FUNCTION_BLOCK FB_LD_PressDemoAuto EXTENDS FB_SequenceBase
VAR
    _partReady, _airReady, _startReady, _stop, _doStep, _processed, _endCycle, _dummy : BOOL;
    _dwellTwoHandHeld : BOOL;          // N220 named wait: two-hand held through the dwell
    _decisionRequest : ST_DecisionRequest;   // §6.11 not-reached confirmation
    _answer : INT;
    _ramReached, _failureConfirmed : BOOL;   // N200/N210 named waits
    _twoHandHeldDuringClose : BOOL;          // N180 named wait
    _closeAbortWarned : BOOL;                // N180 §6.9(e) message result
    _ramFailureReported : BOOL;              // N200 §6.9(e) message result
    _partInMachine : BOOL;                   // §3.16.3 the part is already received
    _partDispositioned : BOOL;               // N260 already set the verdict
    _traceAccepted, _recordAccepted, _partProcessed : BOOL;
    {attribute 'OPC.UA.DA' := '0'}
    _pressRam : REFERENCE TO FB_CylinderCM;
    {attribute 'OPC.UA.DA' := '0'}
    _door : REFERENCE TO FB_CylinderCM;
    {attribute 'OPC.UA.DA' := '0'}
    _partSlide : REFERENCE TO FB_CylinderCM;
    {attribute 'OPC.UA.DA' := '0'}
    _twoHand : REFERENCE TO FB_TwoHandStartCM;
    {attribute 'OPC.UA.DA' := '0'}
    _partPresentSensor : REFERENCE TO FB_DigitalInputCM;
    {attribute 'OPC.UA.DA' := '0'}
    _airPressureMonitor : REFERENCE TO FB_AirPressureMonitorCM;
    {attribute 'OPC.UA.DA' := '0'}
    _parCfg : REFERENCE TO ST_PneumaticPressParCfg;
    // §3.8a - the cell's own policy, referenced like _parCfg.
    {attribute 'OPC.UA.DA' := '0'}
    _stationCfg : REFERENCE TO ST_PneumaticPressStationCfg;
    {attribute 'OPC.UA.DA' := '0'}
    _outCmd : REFERENCE TO ST_PneumaticPressOutCmd;
    {attribute 'OPC.UA.DA' := '0'}
    _startLatched : REFERENCE TO BOOL;
    {attribute 'OPC.UA.DA' := '0'}
    _loadPosition : FB_PressDemoLoadPosition;
END_VAR
VAR // added by the converter: edge detectors and wires of the graphical bodies
    _w1, _w2, _w3, _w4, _w5, _w6, _w7, _w8, _w9, _w10, _w11, _w12, _w13, _w14, _w15, _w16, _w17, _w18, _w19, _w20, _w21, _w22, _w23, _w24, _w25, _w26, _w27, _w28, _w29, _w30 : BOOL;
END_VAR

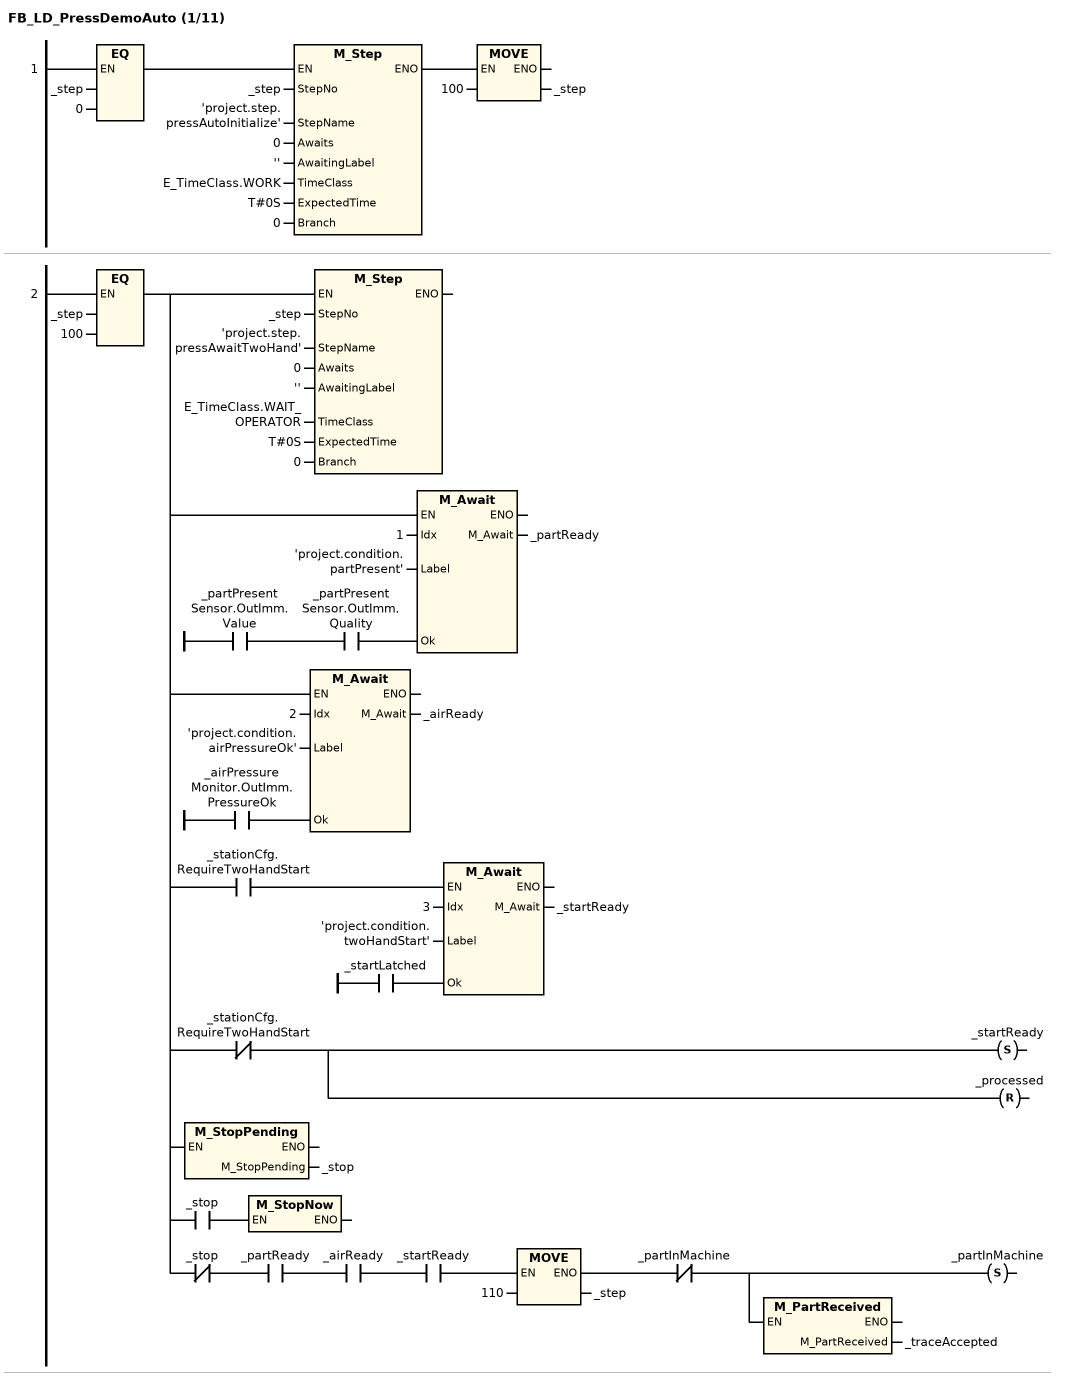
// NETWORK 1
_w1 := _step = 0;
IF _w1 THEN
    M_Step(StepNo := _step, StepName := 'project.step.pressAutoInitialize', Awaits := 0, AwaitingLabel := '', TimeClass := E_TimeClass.WORK, ExpectedTime := T#0S, Branch := 0);
END_IF
IF _w1 THEN _step := 100; END_IF

// NETWORK 2
_w2 := _step = 100;
IF _w2 THEN
    M_Step(StepNo := _step, StepName := 'project.step.pressAwaitTwoHand', Awaits := 0, AwaitingLabel := '', TimeClass := E_TimeClass.WAIT_OPERATOR, ExpectedTime := T#0S, Branch := 0);
END_IF
IF _w2 THEN
    _partReady := M_Await(Idx := 1, Label := 'project.condition.partPresent', Ok := _partPresentSensor.OutImm.Value AND _partPresentSensor.OutImm.Quality);
END_IF
IF _w2 THEN
    _airReady := M_Await(Idx := 2, Label := 'project.condition.airPressureOk', Ok := _airPressureMonitor.OutImm.PressureOk);
END_IF
IF _w2 AND _stationCfg.RequireTwoHandStart THEN
    _startReady := M_Await(Idx := 3, Label := 'project.condition.twoHandStart', Ok := _startLatched);
END_IF
_w3 := _w2 AND NOT _stationCfg.RequireTwoHandStart;
_startReady S= _w3;
_processed R= _w3;
IF _w2 THEN _stop := M_StopPending(); END_IF
IF _w2 AND _stop THEN M_StopNow(); END_IF
IF _w2 AND NOT _stop AND _partReady AND _airReady AND _startReady THEN _step := 110; END_IF
_w4 := (_w2 AND NOT _stop AND _partReady AND _airReady AND _startReady) AND NOT _partInMachine;
_partInMachine S= _w4;
IF _w4 THEN _traceAccepted := M_PartReceived(); END_IF

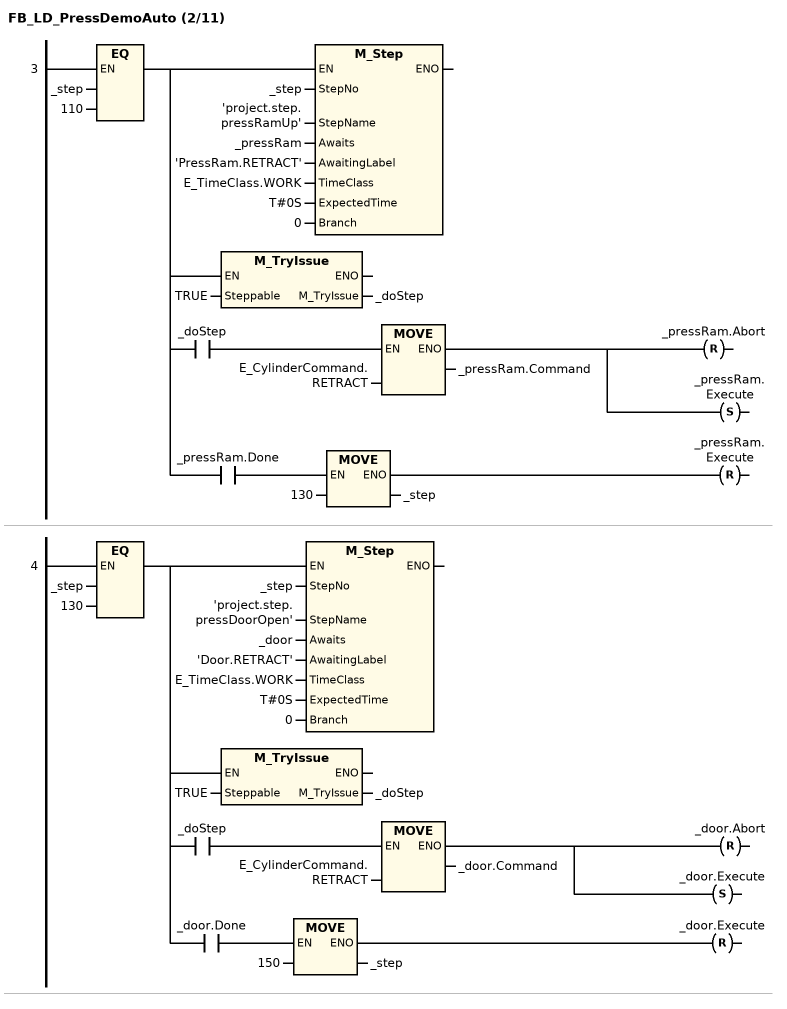
// NETWORK 3
_w5 := _step = 110;
IF _w5 THEN
    M_Step(StepNo := _step, StepName := 'project.step.pressRamUp', Awaits := _pressRam, AwaitingLabel := 'PressRam.RETRACT', TimeClass := E_TimeClass.WORK, ExpectedTime := T#0S, Branch := 0);
END_IF
IF _w5 THEN _doStep := M_TryIssue(Steppable := TRUE); END_IF
IF _w5 AND _doStep THEN _pressRam.Command := E_CylinderCommand.RETRACT; END_IF
_w6 := _w5 AND _doStep;
_pressRam.Abort R= _w6;
_pressRam.Execute S= _w6;
IF _w5 AND _pressRam.Done THEN _step := 130; END_IF
_pressRam.Execute R= _w5 AND _pressRam.Done;

// NETWORK 4
_w7 := _step = 130;
IF _w7 THEN
    M_Step(StepNo := _step, StepName := 'project.step.pressDoorOpen', Awaits := _door, AwaitingLabel := 'Door.RETRACT', TimeClass := E_TimeClass.WORK, ExpectedTime := T#0S, Branch := 0);
END_IF
IF _w7 THEN _doStep := M_TryIssue(Steppable := TRUE); END_IF
IF _w7 AND _doStep THEN _door.Command := E_CylinderCommand.RETRACT; END_IF
_w8 := _w7 AND _doStep;
_door.Abort R= _w8;
_door.Execute S= _w8;
IF _w7 AND _door.Done THEN _step := 150; END_IF
_door.Execute R= _w7 AND _door.Done;

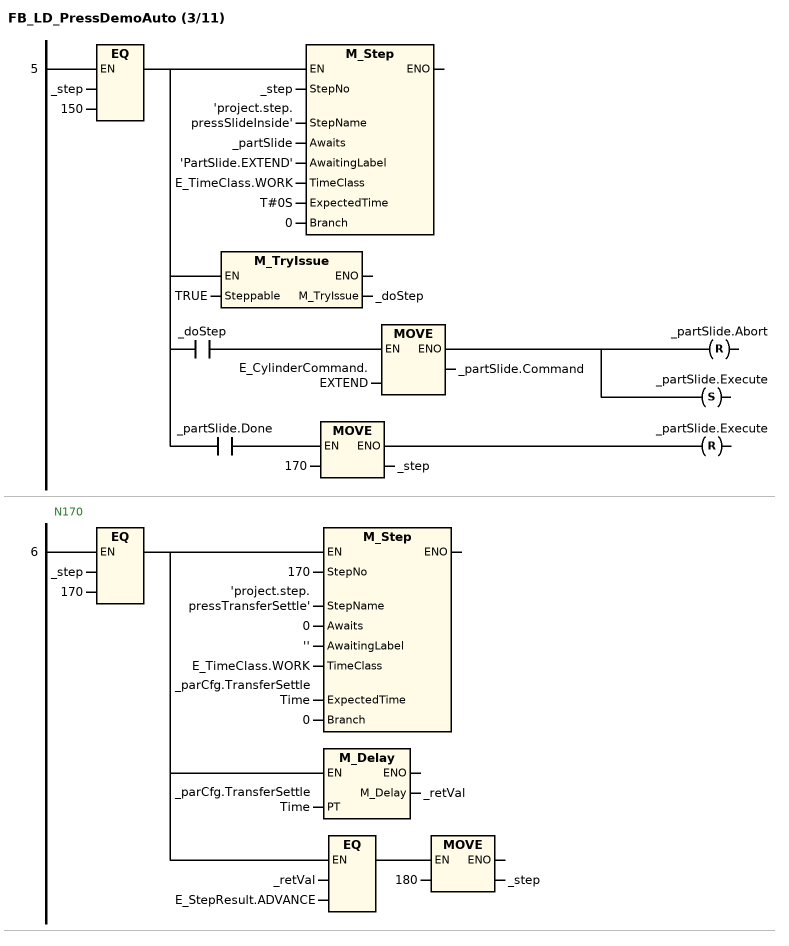
// NETWORK 5
_w9 := _step = 150;
IF _w9 THEN
    M_Step(StepNo := _step, StepName := 'project.step.pressSlideInside', Awaits := _partSlide, AwaitingLabel := 'PartSlide.EXTEND', TimeClass := E_TimeClass.WORK, ExpectedTime := T#0S, Branch := 0);
END_IF
IF _w9 THEN _doStep := M_TryIssue(Steppable := TRUE); END_IF
IF _w9 AND _doStep THEN _partSlide.Command := E_CylinderCommand.EXTEND; END_IF
_w10 := _w9 AND _doStep;
_partSlide.Abort R= _w10;
_partSlide.Execute S= _w10;
IF _w9 AND _partSlide.Done THEN _step := 170; END_IF
_partSlide.Execute R= _w9 AND _partSlide.Done;

// NETWORK 6
// N170
_w11 := _step = 170;
IF _w11 THEN
    M_Step(StepNo := 170, StepName := 'project.step.pressTransferSettle', Awaits := 0, AwaitingLabel := '', TimeClass := E_TimeClass.WORK, ExpectedTime := _parCfg.TransferSettleTime, Branch := 0);
END_IF
IF _w11 THEN _retVal := M_Delay(PT := _parCfg.TransferSettleTime); END_IF
IF _w11 AND _retVal = E_StepResult.ADVANCE THEN _step := 180; END_IF

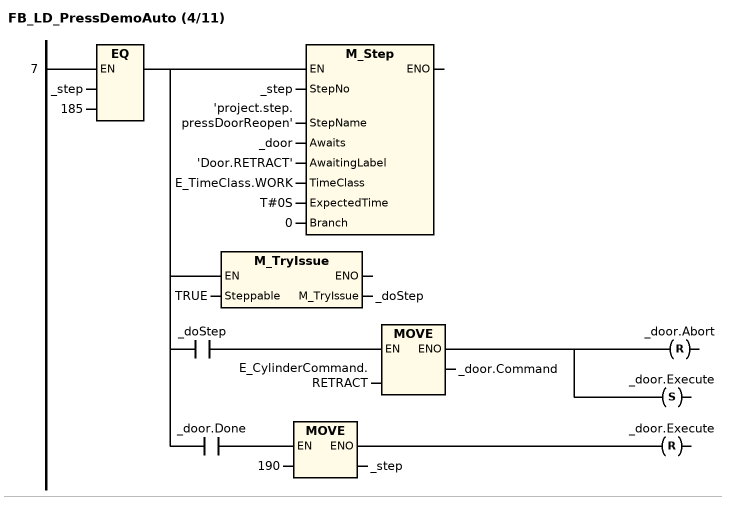
// NETWORK 7
_w12 := _step = 185;
IF _w12 THEN
    M_Step(StepNo := _step, StepName := 'project.step.pressDoorReopen', Awaits := _door, AwaitingLabel := 'Door.RETRACT', TimeClass := E_TimeClass.WORK, ExpectedTime := T#0S, Branch := 0);
END_IF
IF _w12 THEN _doStep := M_TryIssue(Steppable := TRUE); END_IF
IF _w12 AND _doStep THEN _door.Command := E_CylinderCommand.RETRACT; END_IF
_w13 := _w12 AND _doStep;
_door.Abort R= _w13;
_door.Execute S= _w13;
IF _w12 AND _door.Done THEN _step := 190; END_IF
_door.Execute R= _w12 AND _door.Done;

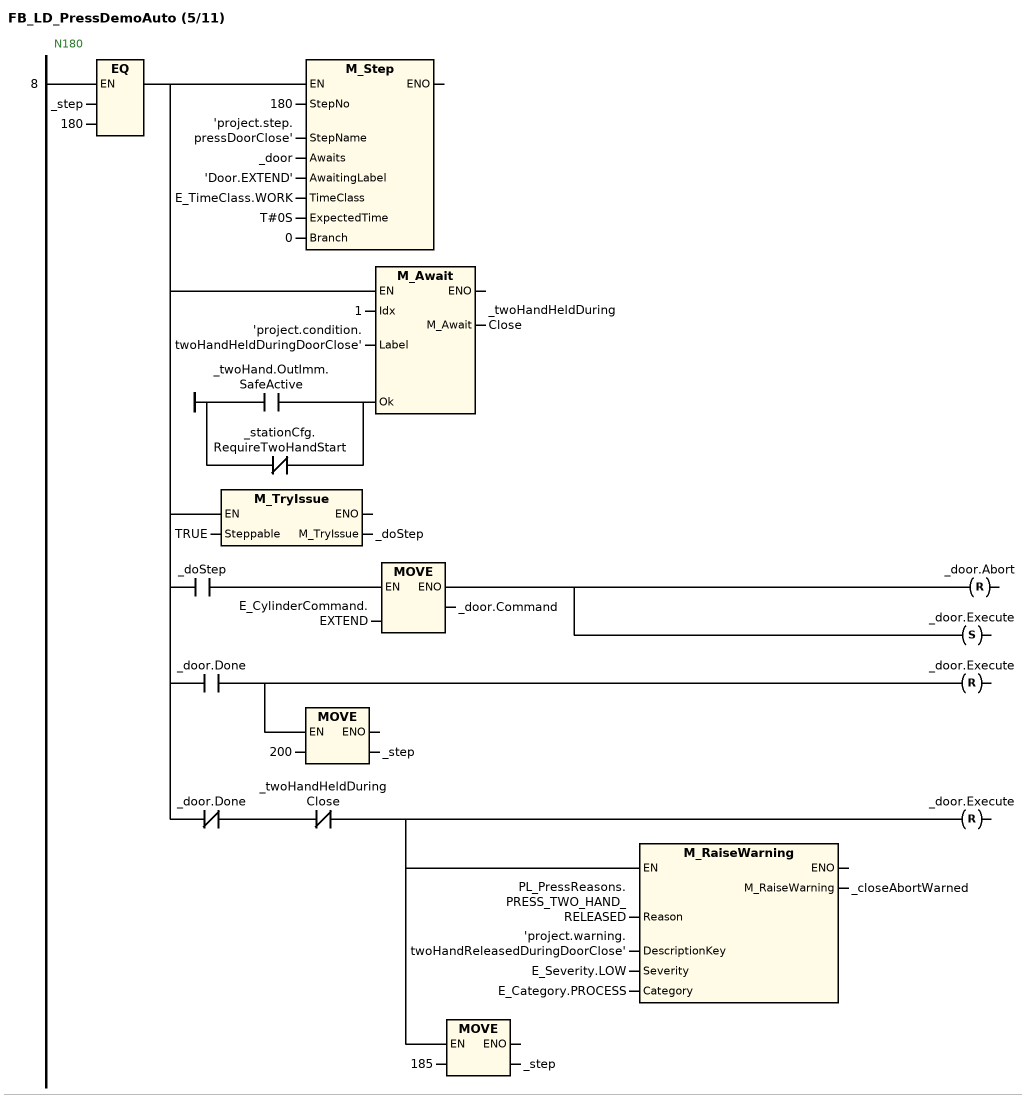
// NETWORK 8
// N180
_w14 := _step = 180;
IF _w14 THEN
    M_Step(StepNo := 180, StepName := 'project.step.pressDoorClose', Awaits := _door, AwaitingLabel := 'Door.EXTEND', TimeClass := E_TimeClass.WORK, ExpectedTime := T#0S, Branch := 0);
END_IF
IF _w14 THEN
    _twoHandHeldDuringClose := M_Await(Idx := 1, Label := 'project.condition.twoHandHeldDuringDoorClose', Ok := _twoHand.OutImm.SafeActive OR NOT _stationCfg.RequireTwoHandStart);
END_IF
IF _w14 THEN _doStep := M_TryIssue(Steppable := TRUE); END_IF
IF _w14 AND _doStep THEN _door.Command := E_CylinderCommand.EXTEND; END_IF
_w15 := _w14 AND _doStep;
_door.Abort R= _w15;
_door.Execute S= _w15;
_w16 := _w14 AND _door.Done;
_door.Execute R= _w16;
IF _w16 THEN _step := 200; END_IF
_w17 := _w14 AND NOT _door.Done AND NOT _twoHandHeldDuringClose;
_door.Execute R= _w17;
IF _w17 THEN
    _closeAbortWarned := M_RaiseWarning(Reason := PL_PressReasons.PRESS_TWO_HAND_RELEASED, DescriptionKey := 'project.warning.twoHandReleasedDuringDoorClose', Severity := E_Severity.LOW, Category := E_Category.PROCESS);
END_IF
IF _w17 THEN _step := 185; END_IF

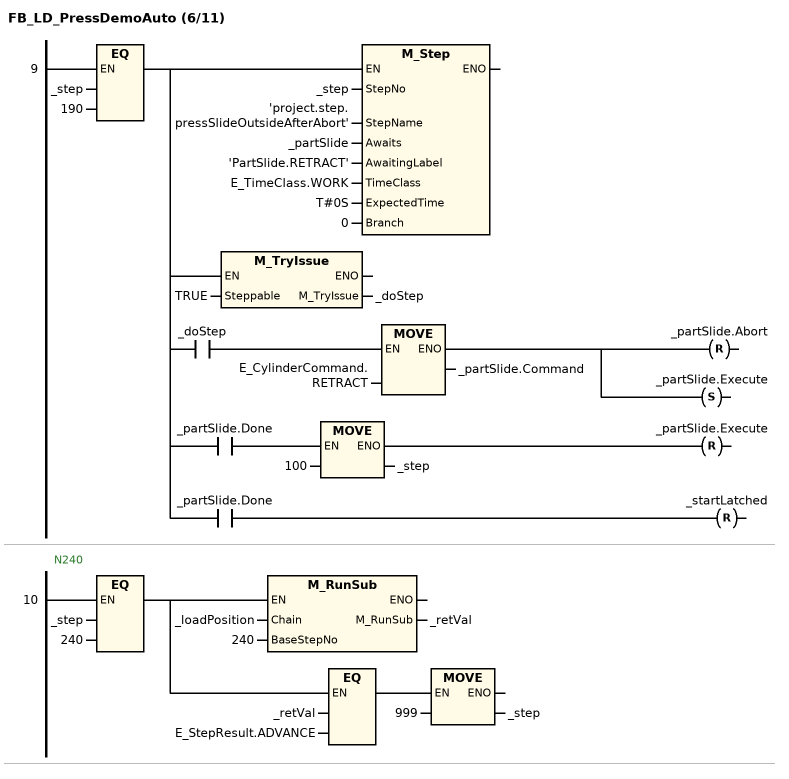
// NETWORK 9
_w18 := _step = 190;
IF _w18 THEN
    M_Step(StepNo := _step, StepName := 'project.step.pressSlideOutsideAfterAbort', Awaits := _partSlide, AwaitingLabel := 'PartSlide.RETRACT', TimeClass := E_TimeClass.WORK, ExpectedTime := T#0S, Branch := 0);
END_IF
IF _w18 THEN _doStep := M_TryIssue(Steppable := TRUE); END_IF
IF _w18 AND _doStep THEN _partSlide.Command := E_CylinderCommand.RETRACT; END_IF
_w19 := _w18 AND _doStep;
_partSlide.Abort R= _w19;
_partSlide.Execute S= _w19;
IF _w18 AND _partSlide.Done THEN _step := 100; END_IF
_partSlide.Execute R= _w18 AND _partSlide.Done;
_startLatched R= _w18 AND _partSlide.Done;

// NETWORK 10
// N240
_w20 := _step = 240;
IF _w20 THEN _retVal := M_RunSub(Chain := _loadPosition, BaseStepNo := 240); END_IF
IF _w20 AND _retVal = E_StepResult.ADVANCE THEN _step := 999; END_IF

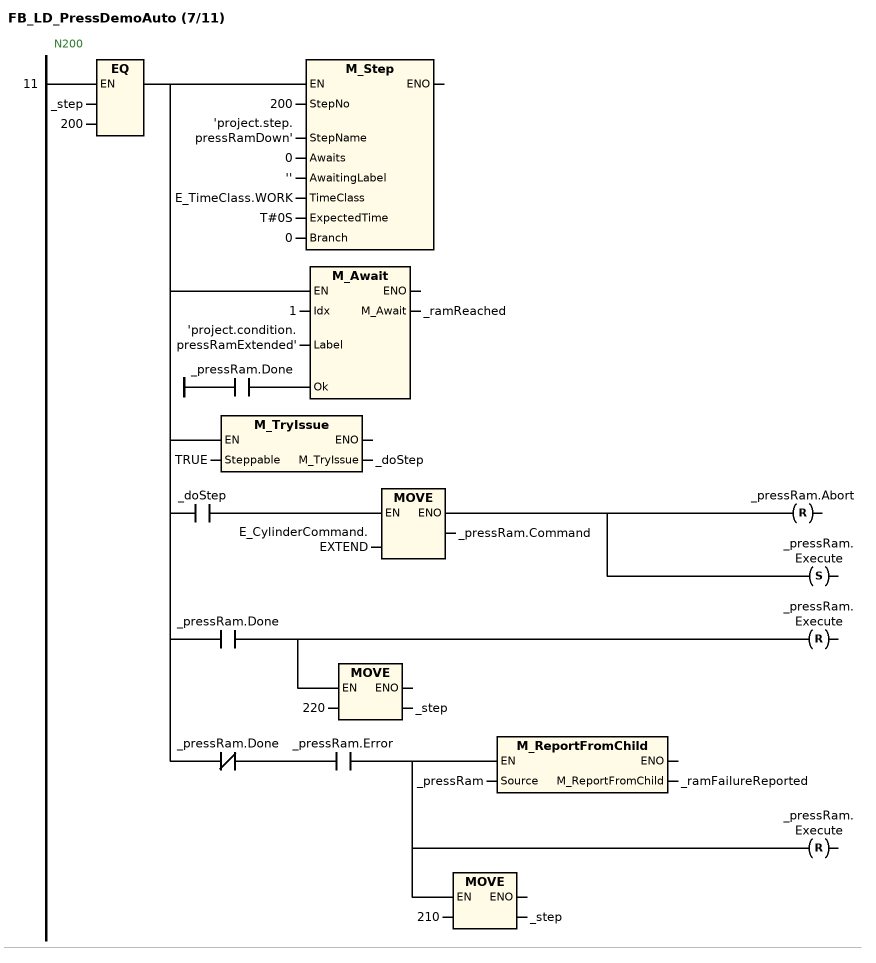
// NETWORK 11
// N200
_w21 := _step = 200;
IF _w21 THEN
    M_Step(StepNo := 200, StepName := 'project.step.pressRamDown', Awaits := 0, AwaitingLabel := '', TimeClass := E_TimeClass.WORK, ExpectedTime := T#0S, Branch := 0);
END_IF
IF _w21 THEN
    _ramReached := M_Await(Idx := 1, Label := 'project.condition.pressRamExtended', Ok := _pressRam.Done);
END_IF
IF _w21 THEN _doStep := M_TryIssue(Steppable := TRUE); END_IF
IF _w21 AND _doStep THEN _pressRam.Command := E_CylinderCommand.EXTEND; END_IF
_w22 := _w21 AND _doStep;
_pressRam.Abort R= _w22;
_pressRam.Execute S= _w22;
_w23 := _w21 AND _pressRam.Done;
_pressRam.Execute R= _w23;
IF _w23 THEN _step := 220; END_IF
_w24 := _w21 AND NOT _pressRam.Done AND _pressRam.Error;
IF _w24 THEN _ramFailureReported := M_ReportFromChild(Source := _pressRam); END_IF
_pressRam.Execute R= _w24;
IF _w24 THEN _step := 210; END_IF

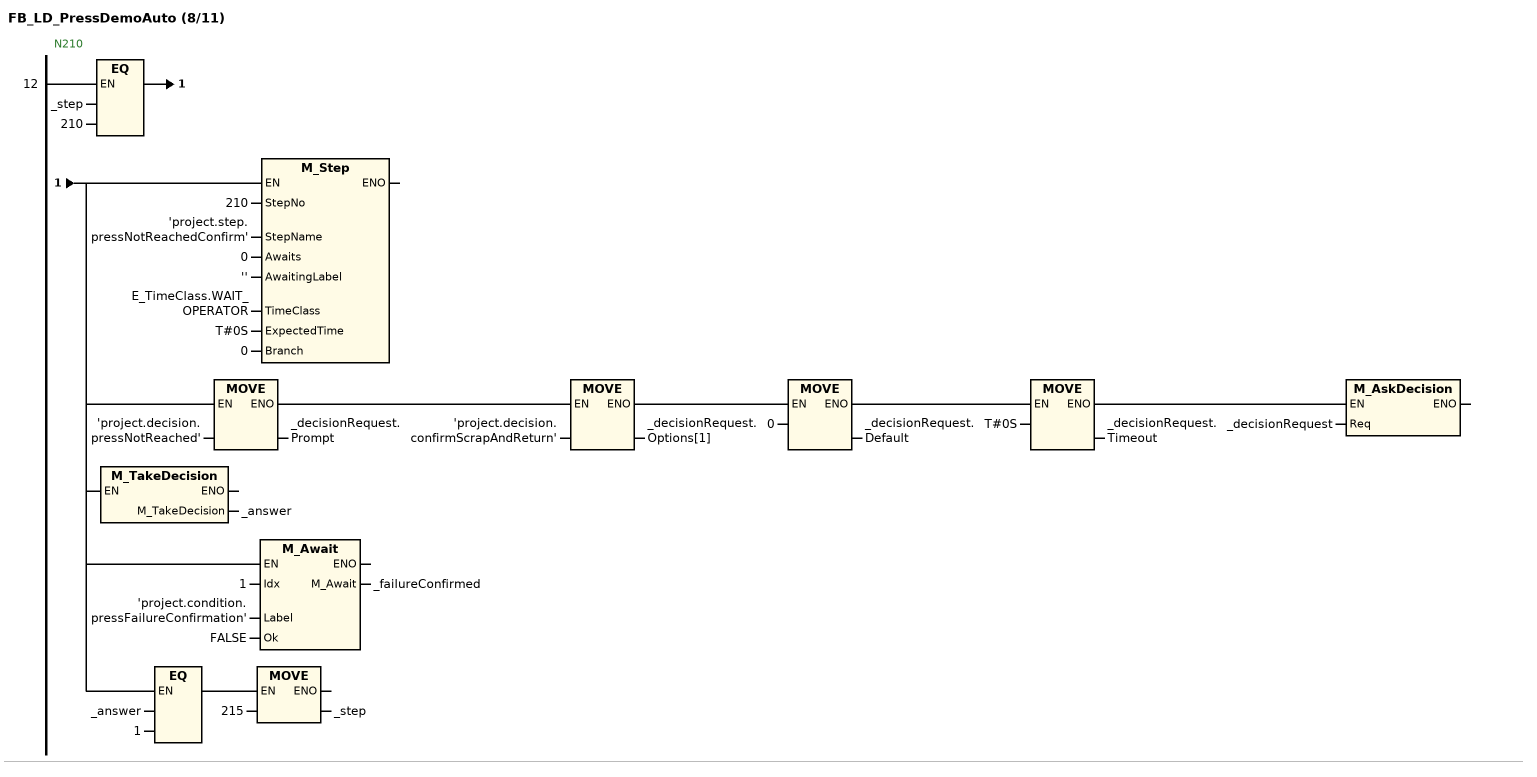
// NETWORK 12
// N210
_w25 := _step = 210;
IF _w25 THEN
    M_Step(StepNo := 210, StepName := 'project.step.pressNotReachedConfirm', Awaits := 0, AwaitingLabel := '', TimeClass := E_TimeClass.WAIT_OPERATOR, ExpectedTime := T#0S, Branch := 0);
END_IF
IF _w25 THEN _decisionRequest.Prompt := 'project.decision.pressNotReached'; END_IF
IF _w25 THEN _decisionRequest.Options[1] := 'project.decision.confirmScrapAndReturn'; END_IF
IF _w25 THEN _decisionRequest.Default := 0; END_IF
IF _w25 THEN _decisionRequest.Timeout := T#0S; END_IF
IF _w25 THEN M_AskDecision(Req := _decisionRequest); END_IF
IF _w25 THEN _answer := M_TakeDecision(); END_IF
IF _w25 THEN
    _failureConfirmed := M_Await(Idx := 1, Label := 'project.condition.pressFailureConfirmation', Ok := FALSE);
END_IF
IF _w25 AND _answer = 1 THEN _step := 215; END_IF

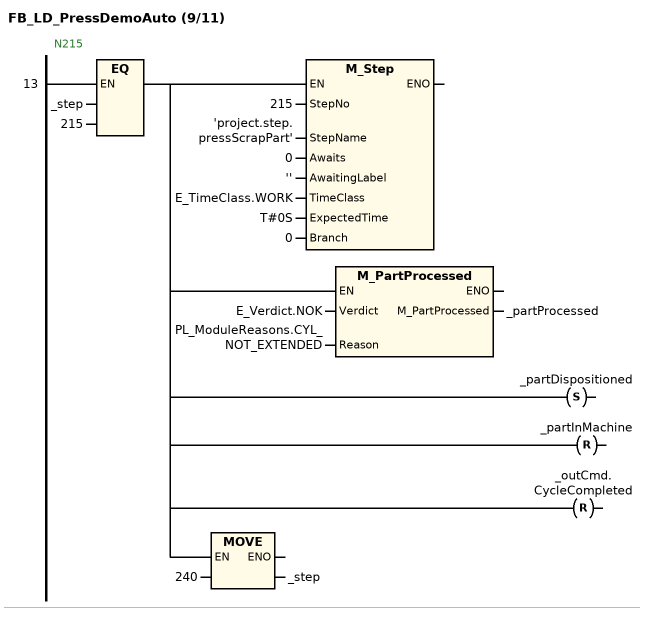
// NETWORK 13
// N215
_w26 := _step = 215;
IF _w26 THEN
    M_Step(StepNo := 215, StepName := 'project.step.pressScrapPart', Awaits := 0, AwaitingLabel := '', TimeClass := E_TimeClass.WORK, ExpectedTime := T#0S, Branch := 0);
END_IF
IF _w26 THEN
    _partProcessed := M_PartProcessed(Verdict := E_Verdict.NOK, Reason := PL_ModuleReasons.CYL_NOT_EXTENDED);
END_IF
_partDispositioned S= _w26;
_partInMachine R= _w26;
_outCmd.CycleCompleted R= _w26;
IF _w26 THEN _step := 240; END_IF

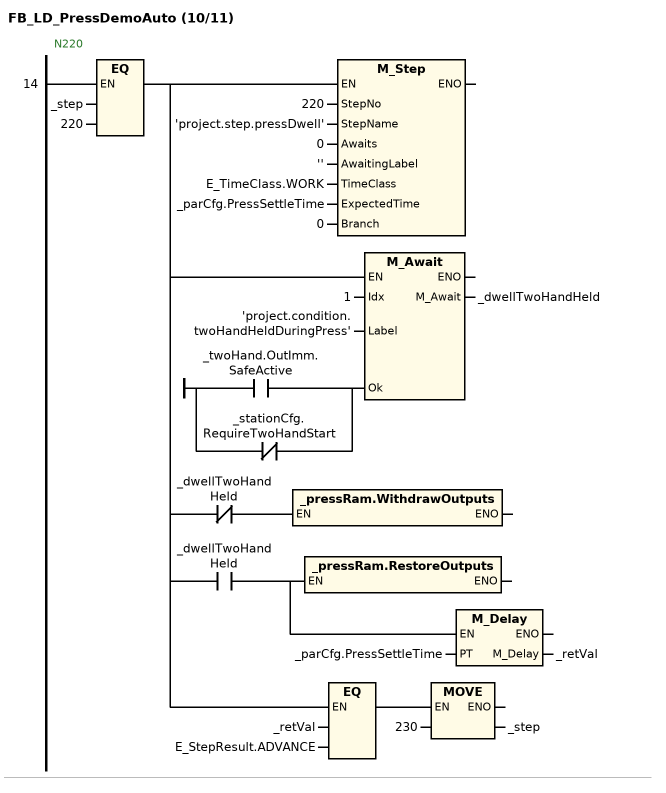
// NETWORK 14
// N220
_w27 := _step = 220;
IF _w27 THEN
    M_Step(StepNo := 220, StepName := 'project.step.pressDwell', Awaits := 0, AwaitingLabel := '', TimeClass := E_TimeClass.WORK, ExpectedTime := _parCfg.PressSettleTime, Branch := 0);
END_IF
IF _w27 THEN
    _dwellTwoHandHeld := M_Await(Idx := 1, Label := 'project.condition.twoHandHeldDuringPress', Ok := _twoHand.OutImm.SafeActive OR NOT _stationCfg.RequireTwoHandStart);
END_IF
IF _w27 AND NOT _dwellTwoHandHeld THEN _pressRam.WithdrawOutputs(); END_IF
_w28 := _w27 AND _dwellTwoHandHeld;
IF _w28 THEN _pressRam.RestoreOutputs(); END_IF
IF _w28 THEN _retVal := M_Delay(PT := _parCfg.PressSettleTime); END_IF
IF _w27 AND _retVal = E_StepResult.ADVANCE THEN _step := 230; END_IF

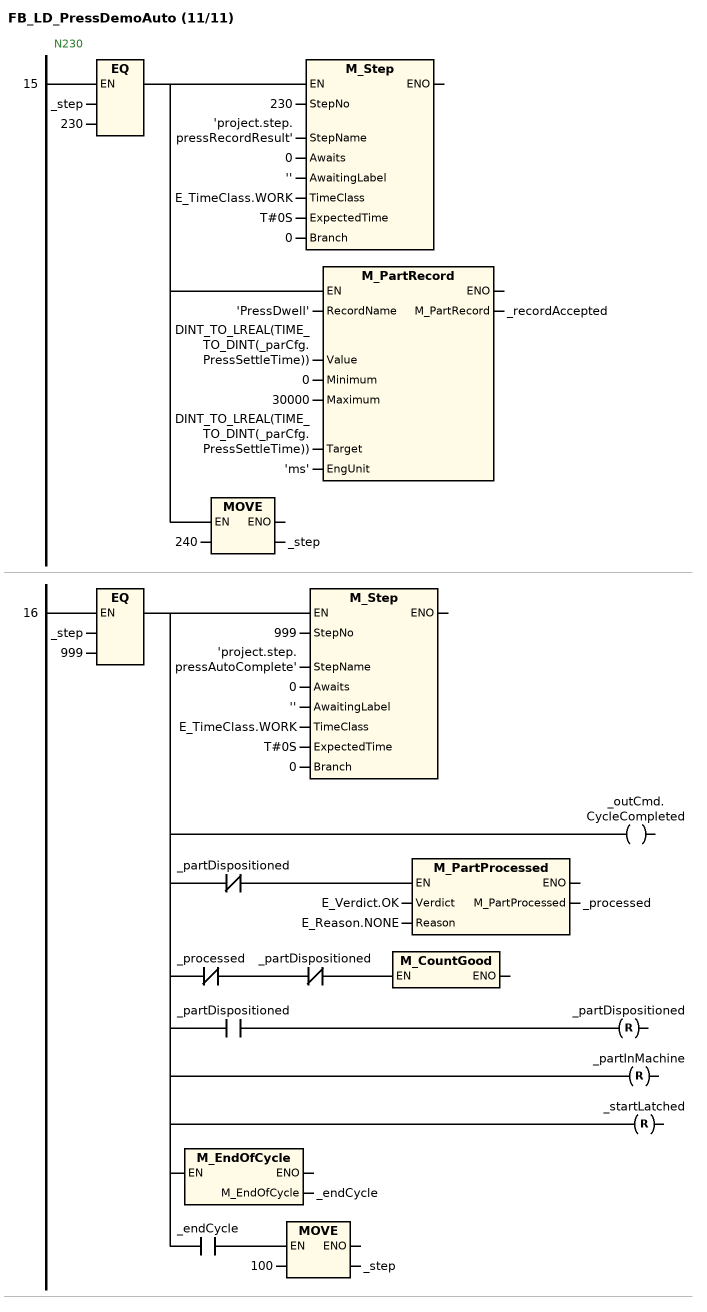
// NETWORK 15
// N230
_w29 := _step = 230;
IF _w29 THEN
    M_Step(StepNo := 230, StepName := 'project.step.pressRecordResult', Awaits := 0, AwaitingLabel := '', TimeClass := E_TimeClass.WORK, ExpectedTime := T#0S, Branch := 0);
END_IF
IF _w29 THEN
    _recordAccepted := M_PartRecord(RecordName := 'PressDwell', Value := DINT_TO_LREAL(TIME_TO_DINT(_parCfg.PressSettleTime)), Minimum := 0, Maximum := 30000, Target := DINT_TO_LREAL(TIME_TO_DINT(_parCfg.PressSettleTime)), EngUnit := 'ms');
END_IF
IF _w29 THEN _step := 240; END_IF

// NETWORK 16
_w30 := _step = 999;
IF _w30 THEN
    M_Step(StepNo := 999, StepName := 'project.step.pressAutoComplete', Awaits := 0, AwaitingLabel := '', TimeClass := E_TimeClass.WORK, ExpectedTime := T#0S, Branch := 0);
END_IF
_outCmd.CycleCompleted := _w30;
IF _w30 AND NOT _partDispositioned THEN
    _processed := M_PartProcessed(Verdict := E_Verdict.OK, Reason := E_Reason.NONE);
END_IF
IF _w30 AND NOT _processed AND NOT _partDispositioned THEN M_CountGood(); END_IF
_partDispositioned R= _w30 AND _partDispositioned;
_partInMachine R= _w30;
_startLatched R= _w30;
IF _w30 THEN _endCycle := M_EndOfCycle(); END_IF
IF _w30 AND _endCycle THEN _step := 100; END_IF

// Identical signature to the ST and SFC renditions of this chain, so the Unit can
// bind whichever one AUTO_SEQUENCE_LANGUAGE selects without any other difference.
METHOD Setup : BOOL
VAR_INPUT
    Host : I_SequenceHost;
END_VAR
VAR_IN_OUT
    PressRam : FB_CylinderCM;
    Door : FB_CylinderCM;
    PartSlide : FB_CylinderCM;
    TwoHand : FB_TwoHandStartCM;
    PartPresentSensor : FB_DigitalInputCM;
    AirPressureMonitor : FB_AirPressureMonitorCM;
    ParCfg : ST_PneumaticPressParCfg;
    StationCfg : ST_PneumaticPressStationCfg;
    OutCmd : ST_PneumaticPressOutCmd;
    StartLatched : BOOL;
END_VAR
_pressRam REF= PressRam;
_door REF= Door;
_partSlide REF= PartSlide;
_twoHand REF= TwoHand;
_partPresentSensor REF= PartPresentSensor;
_airPressureMonitor REF= AirPressureMonitor;
_parCfg REF= ParCfg;
_stationCfg REF= StationCfg;
_outCmd REF= OutCmd;
_startLatched REF= StartLatched;
Setup := M_Attach(Host := Host) AND __ISVALIDREF(_pressRam) AND __ISVALIDREF(_door)
    AND __ISVALIDREF(_partSlide) AND __ISVALIDREF(_twoHand)
    AND __ISVALIDREF(_partPresentSensor) AND __ISVALIDREF(_airPressureMonitor)
    AND __ISVALIDREF(_parCfg) AND __ISVALIDREF(_outCmd) AND __ISVALIDREF(_startLatched)
    AND _loadPosition.Setup(Host := Host, PressRam := PressRam, Door := Door, PartSlide := PartSlide);
END_METHOD

METHOD M_Reset
M_ResetBase(0);
// A chart reset abandons whatever the cycle was holding: the part record is
// closed by N215/N999, never by a reset, so both trackers start clean.
_partDispositioned := FALSE;
_partInMachine := FALSE;
END_METHOD

END_FUNCTION_BLOCK

(* stored: Version 1.1.0.1
   POU FB_LD_PressDemoAuto: Id {3dfbbe8c-f8a4-4989-8f97-e499328e9847}, SpecialFunc None
   Method Setup: Id {9f2c41ab-73d5-4e18-9c60-2ad4f1e77b31}
   Method M_Reset: Id {4c1e8b02-59d7-4a63-b8f1-6e0d92c3aa17} *)
